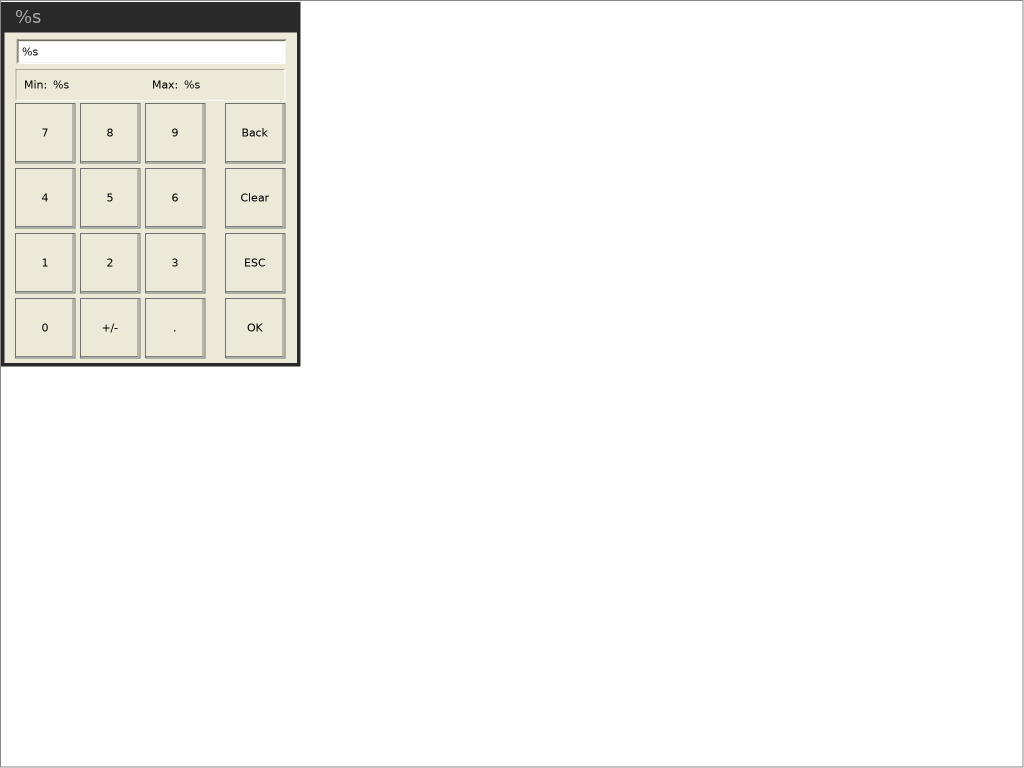
VISUALIZATION Numpad  // 1024x768
VAR_INPUT
	stVariableValue : STRING;
	stMin : STRING;
	stMax : STRING;
	wstTitle : WSTRING;
	flags : DWORD;
END_VAR
VAR
	bInit : BOOL;
	stMessage : STRING;
	stOutputValue : STRING;
	iCaretPosition	: INT;
	iSelectionStart	: INT;
	iSelectionEnd	: INT;
	xAllSelected	: BOOL;
END_VAR
    Rectangle (3,31 294x39)
    Polyline (17,63) (17,39) (286,39)
    Polyline (18,63) (285,63) (285,40)
    Polyline (18,62) (18,40) (285,40)
    Textfield (19,42 265x20), "%s", text variable: stOutputValue
        p905179711: iCaretPosition
        p3815007873: iSelectionStart
        p1425650380: iSelectionEnd
        p3479897389: xAllSelected
    Rectangle (3,98 295x67)
    Rectangle (3,165 295x65)
    Rectangle (3,230 295x65)
    Rectangle (3,295 295x68)
    Button (225,298 60x60), "OK"
        OnMouseDown: CloseDialog Dialog=Numpad, Result=OK, NumpadKeypad=True, NumpadKeypadSet=True
    Button (225,233 60x60), "ESC"
        OnMouseDown: CloseDialog Dialog=Numpad, Result=Cancel, NumpadKeypad=True, NumpadKeypadSet=True
    Button (225,168 60x60), "Clear"
        OnMouseDown: execute {
            stVariableValue := '';
            stOutputValue := '';
            flags := flags AND NOT 16#0008;
            flags := flags AND NOT 16#0010;
            iCaretPosition	:= 1;
            iSelectionStart	:= 1;
            iSelectionEnd	:= 1;
        }
    Button (225,103 60x60), "Back"
        OnMouseDown: execute { VisuDlg_ProcessBack(stOutputValue, stVariableValue, iCaretPosition, iSelectionStart, iSelectionEnd, bInit); }
    Button (145,298 60x60), "."
        OnMouseDown: execute { VisuDlg_ProcessChar(stOutputValue, stVariableValue, iCaretPosition, iSelectionStart, iSelectionEnd, (flags AND VisuElems.Visu_InputFlags.Password) = 1, '.'); }
    Button (80,298 60x60), "+/-"
        OnMouseDown: execute { VisuDlg_ProcessChangeSign(stOutputValue, stVariableValue, iCaretPosition, iSelectionStart, iSelectionEnd, (flags AND VisuElems.Visu_InputFlags.Password) = 1); }
    Button (15,298 60x60), "0"
        OnMouseDown: execute { VisuDlg_ProcessChar(stOutputValue, stVariableValue, iCaretPosition, iSelectionStart, iSelectionEnd, (flags AND VisuElems.Visu_InputFlags.Password) = 1, '0'); }
    Button (15,233 60x60), "1"
        OnMouseDown: execute { VisuDlg_ProcessChar(stOutputValue, stVariableValue, iCaretPosition, iSelectionStart, iSelectionEnd, (flags AND VisuElems.Visu_InputFlags.Password) = 1, '1'); }
    Button (80,233 60x60), "2"
        OnMouseDown: execute { VisuDlg_ProcessChar(stOutputValue, stVariableValue, iCaretPosition, iSelectionStart, iSelectionEnd, (flags AND VisuElems.Visu_InputFlags.Password) = 1, '2'); }
    Button (145,233 60x60), "3"
        OnMouseDown: execute { VisuDlg_ProcessChar(stOutputValue, stVariableValue, iCaretPosition, iSelectionStart, iSelectionEnd, (flags AND VisuElems.Visu_InputFlags.Password) = 1, '3'); }
    Button (15,168 60x60), "4"
        OnMouseDown: execute { VisuDlg_ProcessChar(stOutputValue, stVariableValue, iCaretPosition, iSelectionStart, iSelectionEnd, (flags AND VisuElems.Visu_InputFlags.Password) = 1, '4'); }
    Button (80,168 60x60), "5"
        OnMouseDown: execute { VisuDlg_ProcessChar(stOutputValue, stVariableValue, iCaretPosition, iSelectionStart, iSelectionEnd, (flags AND VisuElems.Visu_InputFlags.Password) = 1, '5'); }
    Button (145,168 60x60), "6"
        OnMouseDown: execute { VisuDlg_ProcessChar(stOutputValue, stVariableValue, iCaretPosition, iSelectionStart, iSelectionEnd, (flags AND VisuElems.Visu_InputFlags.Password) = 1, '6'); }
    Button (15,103 60x60), "7"
        OnMouseDown: execute { VisuDlg_ProcessChar(stOutputValue, stVariableValue, iCaretPosition, iSelectionStart, iSelectionEnd, (flags AND VisuElems.Visu_InputFlags.Password) = 1, '7'); }
    Button (80,103 60x60), "8"
        OnMouseDown: execute { VisuDlg_ProcessChar(stOutputValue, stVariableValue, iCaretPosition, iSelectionStart, iSelectionEnd, (flags AND VisuElems.Visu_InputFlags.Password) = 1, '8'); }
    Button (145,103 60x60), "9"
        OnMouseDown: execute { VisuDlg_ProcessChar(stOutputValue, stVariableValue, iCaretPosition, iSelectionStart, iSelectionEnd, (flags AND VisuElems.Visu_InputFlags.Password) = 1, '9'); }
    Rectangle (3,69 294x33)
    Rectangle (50,75 95x20), "%s", text variable: stMin, invisible if: LEN(stMin) = 0
        p55702900: SEL(((UDINT_TO_DINT(flags AND 16#0008))=16#0008),16#FF000000,16#FFFF0000)
    Rectangle (181,75 95x20), "%s", text variable: stMax, invisible if: LEN(stMax) = 0
        p55702900: SEL(((UDINT_TO_DINT(flags AND 16#0010))=16#0010),16#FF000000,16#FFFF0000)
    Rectangle (149,75 31x20), "Max:", invisible if: LEN(stMax) = 0
        p55702900: SEL(((UDINT_TO_DINT(flags AND 16#0010))=16#0010),16#FF000000,16#FFFF0000)
    Rectangle (296,363 3x3)
    Rectangle (297,2 3x362)
    Rectangle (1,3 3x360)
    Rectangle (1,2 298x30), invisible if: VisuElems.g_VisualizationStyle.GetDINT('Dialog-UseHeaderColor', 0, 0) = 0
    Rectangle (12,7 280x20), "%s", text variable: gsPadTitle
    Rectangle (1,363 299x3)
    Polyline (16,99) (16,69) (284,69)
    Polyline (17,100) (285,100) (285,69)
    Rectangle (21,75 31x20), "Min:", invisible if: LEN(stMin) = 0
        p55702900: SEL(((UDINT_TO_DINT(flags AND 16#0008))=16#0008),16#FF000000,16#FFFF0000)
END_VISUALIZATION

(* stored: Version 1.1.0.1, ProductVersion 3.1.4024.2
   Visu Numpad: Id {d0bcbbfb-15f4-4b74-bb9b-bcf1302ffd3d} *)
